// TIA Portal V20 export
FUNCTION_BLOCK "FB_IntLoadUnloadOP"   // FB73, SCL
{ S7_Optimized_Access := 'TRUE' }
// stored: AutoNumber false, MemoryReserve 100, SetENOAutomatically false
   VAR_INPUT
      iStartSeqCond : Bool;   // Start Sequence Conditions
      iJobReq : Bool;   // Job Request - From Main
      iShuttleIntLoadUnloadPos : Bool;   // Load/Unload Pos. Reached - Param
      iShuttleIntLoadUnloadPosSetPoint : LReal;   // Load/Unload Pos. Setpoint - Param
      iShuttleIntLoadUnloadOP_Pos : Bool;   // Load/Unload Pos. Reached - Param
      iShuttleIntLoadUnloadOP_PosSetPoint : LReal;   // Load/Unload Pos. Setpoint - Param
      iAxisV_LoadUnloadShuttlePos : Bool;
      iAxisV_LoadUnloadShuttlePosSetPoint : LReal;
      iAxisV_SafePos : Bool;
      iAxisV_SafePosSetPoint : LReal;
      iAxisW_SafePos : Bool;
      iAxisW_SafePosSetPoint : LReal;
      iAxisW_ApproachLoadUnloadPos : Bool;
      iAxisW_ApproachLoadUnloadSetPoint : LReal;
      iAxisW_LoadUnloadPos : Bool;
      iAxisW_LoadUnloadPosSetPoint : LReal;
      iShuttleMoving : Bool;   // Shuttle is moving - From FB_LoaderAxis
      iShuttleInPos : Bool;   // Shuttle pos. reached - From FB_LoaderAxis
      iAxisV_Moving : Bool;   // Shuttle is moving
      iAxisV_InPos : Bool;
      iAxisW_Moving { ExternalAccessible := 'False'; ExternalVisible := 'False'; ExternalWritable := 'False'} : Bool;   // Shuttle is moving
      iAxisW_InPos : Bool;
      iDrilledPartToUnload : Bool;   // Drilled Part To Unload - From FB_Position
      iUnDrilledPartToLoad : Bool;   // Unrilled Part To Load - From FB_Position
      iLoadGripperClosed : Bool;
      iUnloadGripperOpen : Bool;
      iPLC_DateAndTime : DTL;
      iStepPause : Bool;
   END_VAR
   VAR_OUTPUT
      oShuttleStartReq { ExternalAccessible := 'False'; ExternalVisible := 'False'; ExternalWritable := 'False'} : Bool;   // Shuttle Start Order - To FB_LoaderAxis
      oShuttlePosSetPoint { ExternalAccessible := 'False'; ExternalVisible := 'False'; ExternalWritable := 'False'} : Real;   // Shuttle Position Setpoint - To FB_LoaderAxis
      oAxisV_StartReq : Bool;
      oAxisV_PosSetPoint : Real;
      oAxisW_StartReq : Bool;
      oAxisW_PosSetPoint : Real;
      oLoadGripperCloseReq : Bool;
      oUnloadGripperOpenReq : Bool;
   END_VAR
   VAR
      sCurrent_Step_NB : Int;   // Active Step Number
      sCheck_Step_Condition : Bool;
      sOneStepForward : Bool;
      sRTOneStepForward : R_TRIG;
      sOneStepMode { S7_SetPoint := 'True'} : Bool;
      sStepForward : Bool;
      sInterface : "UDT_SequenceInterface";
      sShuttleStartReq { ExternalAccessible := 'False'; ExternalVisible := 'False'; ExternalWritable := 'False'} : Bool;
      sShuttlePosSetPoint { ExternalAccessible := 'False'; ExternalVisible := 'False'; ExternalWritable := 'False'} : Real;
      sAxisV_StartReq : Bool;
      sAxisV_PosSetPoint : Real;
      sAxisW_StartReq : Bool;
      sAxisW_PosSetPoint : Real;
      sLoadGripperCloseReq : Bool;   // Drilled Part To Unload - From FB_Position
      sUnloadGripperOpenReq : Bool;   // Unrilled Part To Load - From FB_Position
      sTimerAfterGripperClose : TON_TIME;
      sTimerAfterGripperOpen : TON_TIME;
      sTimerAfterApproach { S7_SetPoint := 'True'} : TON_TIME;
      sHistory : Struct
         Activation : Bool;
         Steps : Array[0..99] of Int;
         Date_Time : Array[0..99] of DTL;
      END_STRUCT;
      StepText : "FB_GetTextErrorCode";
   END_VAR
   VAR_TEMP
      tIndex : Int;   // Index
   END_VAR
   VAR CONSTANT
      S00_INIT : Int := 0;
      S10_CHECK_INT_LOAD_UNLOAD_OPTION : Int := 10;
      S20_SHUTTLE_TO_INT_LOAD_UNLOAD_POS_START_REQ : Int := 20;
      S30_SHUTTLE_TO_INT_LOAD_UNLOAD_POS_REACHED : Int := 30;
      S40_AXIS_W_TO_SAFE_POS_START_REQ : Int := 40;
      S50_AXIS_W_TO_SAFE_POS_REACHED : Int := 50;
      S60_AXIS_V_TO_INT_LOAD_UNLOAD_POS_START_REQ : Int := 60;
      S70_AXIS_V_TO_INT_LOAD_UNLOAD_POS_REACHED : Int := 70;
      S80_AXIS_W_TO_INT_LOAD_UNLOAD_APPROACH_POS_START_REQ : Int := 80;
      S90_AXIS_W_TO_INT_LOAD_UNLOAD_APPROACH_POS_REACHED : Int := 90;
      S100_AXIS_W_TO_INT_LOAD_UNLOAD_POS_START_REQ : Int := 100;
      S110_AXIS_W_TO_INT_LOAD_UNLOAD_POS_REACHED : Int := 110;
      S120_CLOSE_LOAD_GRIPPER : Int := 120;
      S130_AXIS_W_TO_SAFE_POS_START_REQ : Int := 130;
      S140_AXIS_W_TO_SAFE_POS_REACHED : Int := 140;
      S150_SHUTTLE_TO_INT_LOAD_UNLOAD_OP_POS_START_REQ : Int := 150;
      S160_SHUTTLE_TO_INT_LOAD_UNLOAD_OP_POS_REACHED : Int := 160;
      S170_AXIS_W_TO_INT_LOAD_UNLOAD_APPROACH_POS_START_REQ : Int := 170;
      S180_AXIS_W_TO_INT_LOAD_UNLOAD_APPROACH_POS_REACHED : Int := 180;
      S190_AXIS_W_TO_INT_LOAD_UNLOAD_POS_START_REQ : Int := 190;
      S200_AXIS_W_TO_INT_LOAD_UNLOAD_POS_REACHED : Int := 200;
      S210_OPEN_UNLOAD_GRIPPER : Int := 210;
      S220_AXIS_W_TO_SAFE_POS_START_REQ : Int := 220;
      S230_AXIS_W_TO_SAFE_POS_REACHED : Int := 230;
      S240_AXIS_V_TO_SAFE_POS_START_REQ : Int := 240;
      S250_AXIS_V_TO_SAFE_POS_REACHED : Int := 250;
      S260_NO_PART_TO_LOAD_UNLOAD : Int := 260;
      S295_JOB_DONE : Int := 295;
   END_VAR
   // StepText.sCode_error[0].ErrorCode := 0;
   // StepText.sCode_error[1].ErrorCode := 10;
   // StepText.sCode_error[2].ErrorCode := 20;
   // StepText.sCode_error[3].ErrorCode := 30;
   // StepText.sCode_error[4].ErrorCode := 40;
   // StepText.sCode_error[5].ErrorCode := 50;
   // StepText.sCode_error[6].ErrorCode := 60;
   // StepText.sCode_error[7].ErrorCode := 70;
   // StepText.sCode_error[8].ErrorCode := 80;
   // StepText.sCode_error[9].ErrorCode := 90;
   // StepText.sCode_error[10].ErrorCode := 95;
BEGIN
   REGION Description header 
       //==================================================================================
       // POSALUX Swiss SA / (C) Copyright 2026
       //----------------------------------------------------------------------------------
       // Title: FB_ExtLoadUnload_OP
       // Comment/Function: 
       // Author: Fabien WALDT
       // Engineering: TIA Portal v20
       //----------------------------------------------------------------------------------
       // Change log table:
       // Version  | Date     | Expert in charge | Changes applied
       // ---------|----------|------------------|-----------------------------------------
       // 00.00.01 | 20260128 | WFA              | First released version
       // =================================================================================
   END_REGION

   REGION Define condition to start
       IF #iStartSeqCond THEN
           #sInterface.SequenceReleased := TRUE;
       ELSE
           // Standard sequencer controls
           #sInterface.SequenceReleased := FALSE;
           #sCurrent_Step_NB := #S00_INIT;
           #sInterface.SequenceRun := FALSE;
           #sInterface.JobDone := FALSE;
           #sCheck_Step_Condition := FALSE;

           // Dedicated sequencer controls
           #sShuttleStartReq := FALSE;
           #sShuttlePosSetPoint := 0.0;
           #sAxisV_StartReq := FALSE;
           #sAxisV_PosSetPoint := 0.0;
           #sAxisW_StartReq := FALSE;
           #sAxisW_PosSetPoint := 0.0;
           #sLoadGripperCloseReq := FALSE;
           #sUnloadGripperOpenReq := FALSE;

           // Add specifics controls 
       END_IF;

       // Reset interface error
       IF #sInterface.Reset THEN
           #sInterface.Error := FALSE;
       END_IF;

       // Reset start when axis in position
       IF #iShuttleInPos THEN
           #sShuttleStartReq := FALSE;
       END_IF;
       IF #iAxisV_InPos THEN
           #sAxisV_StartReq := FALSE;
       END_IF;
       IF #iAxisW_InPos THEN
           #sAxisW_StartReq := FALSE;
       END_IF;

       // One step forward
       #sRTOneStepForward.CLK := #sOneStepForward;
       #sRTOneStepForward();
       #sStepForward := (NOT #sOneStepMode OR (#sOneStepMode AND #sRTOneStepForward.Q)) AND NOT #iStepPause;
       #sOneStepForward := FALSE;

       // Action only true in dedicated steps
       #sLoadGripperCloseReq := FALSE;
       #sUnloadGripperOpenReq := FALSE;

       // Timer Gripper OK
       #"sTimerAfterGripperClose"(IN := #sCurrent_Step_NB = 120
                                  AND ((#iUnDrilledPartToLoad AND #iLoadGripperClosed) OR NOT #iUnDrilledPartToLoad),
                                  PT := T#500ms);
       #"sTimerAfterGripperOpen"(IN := #sCurrent_Step_NB = 210
                                 AND ((#iDrilledPartToUnload AND #iUnloadGripperOpen) OR NOT #iDrilledPartToUnload),
                                 PT := T#500ms);

       // Timer between approach and Load/Unload position
       #sTimerAfterApproach(IN := (#sCurrent_Step_NB = 90 OR #sCurrent_Step_NB = 180) AND #iAxisW_ApproachLoadUnloadPos,
                            PT := T#100ms);
   END_REGION

   REGION Sequence Function
       CASE #sCurrent_Step_NB OF
           #S00_INIT:
               REGION S00 INIT
                   #sCheck_Step_Condition := TRUE;
               END_REGION
           #S10_CHECK_INT_LOAD_UNLOAD_OPTION:
               REGION S10_CHECK_INT_LOAD_UNLOAD_OPTION
                   #sCheck_Step_Condition := TRUE;
               END_REGION
           #S20_SHUTTLE_TO_INT_LOAD_UNLOAD_POS_START_REQ:
               REGION S20_SHUTTLE_TO_INT_LOAD_UNLOAD_POS_START_REQ
                   #sShuttleStartReq := NOT #iShuttleIntLoadUnloadPos;
                   #sShuttlePosSetPoint := LREAL_TO_REAL(#iShuttleIntLoadUnloadPosSetPoint);
                   #sCheck_Step_Condition := TRUE;
               END_REGION
           #S30_SHUTTLE_TO_INT_LOAD_UNLOAD_POS_REACHED:
               REGION S30_SHUTTLE_TO_INT_LOAD_UNLOAD_POS_REACHED
                   #sCheck_Step_Condition := TRUE;
               END_REGION
           #S40_AXIS_W_TO_SAFE_POS_START_REQ:
               REGION S40_AXIS_W_TO_SAFE_POS_START_REQ
                   #sAxisW_StartReq := NOT #iAxisW_SafePos;
                   #sAxisW_PosSetPoint := LREAL_TO_REAL(#iAxisW_SafePosSetPoint);
                   #sCheck_Step_Condition := TRUE;
               END_REGION
           #S50_AXIS_W_TO_SAFE_POS_REACHED:
               REGION S50_AXIS_W_TO_SAFE_POS_REACHED
                   #sCheck_Step_Condition := TRUE;
               END_REGION
           #S60_AXIS_V_TO_INT_LOAD_UNLOAD_POS_START_REQ:
               REGION S60_AXIS_V_TO_INT_LOAD_UNLOAD_POS_START_REQ
                   #sAxisV_StartReq := NOT #iAxisV_LoadUnloadShuttlePos;
                   #sAxisV_PosSetPoint := LREAL_TO_REAL(#iAxisV_LoadUnloadShuttlePosSetPoint);
                       #sCheck_Step_Condition := TRUE;
                   END_REGION
           #S70_AXIS_V_TO_INT_LOAD_UNLOAD_POS_REACHED:
               REGION S70_AXIS_V_TO_INT_LOAD_UNLOAD_POS_REACHED
                   #sCheck_Step_Condition := TRUE;
               END_REGION
           #S80_AXIS_W_TO_INT_LOAD_UNLOAD_APPROACH_POS_START_REQ:
               REGION S80_AXIS_W_TO_INT_LOAD_UNLOAD_APPROACH_POS_START_REQ
                   #sAxisW_StartReq := NOT #iAxisW_ApproachLoadUnloadPos;
                   #sAxisW_PosSetPoint := LREAL_TO_REAL(#iAxisW_ApproachLoadUnloadSetPoint);
                   #sCheck_Step_Condition := TRUE;
               END_REGION
           #S90_AXIS_W_TO_INT_LOAD_UNLOAD_APPROACH_POS_REACHED:
               REGION S90_AXIS_W_TO_INT_LOAD_UNLOAD_APPROACH_POS_REACHED
                   IF #sTimerAfterApproach.Q THEN
                       #sCheck_Step_Condition := TRUE;
                   END_IF;
               END_REGION
           #S100_AXIS_W_TO_INT_LOAD_UNLOAD_POS_START_REQ:
               REGION S100_AXIS_W_TO_INT_LOAD_UNLOAD_POS_START_REQ
                   #sAxisW_StartReq := NOT #iAxisW_LoadUnloadPos;
                   #sAxisW_PosSetPoint := LREAL_TO_REAL(#iAxisW_LoadUnloadPosSetPoint);
                   #sCheck_Step_Condition := TRUE;
               END_REGION
           #S110_AXIS_W_TO_INT_LOAD_UNLOAD_POS_REACHED:
               REGION S110_AXIS_W_TO_INT_LOAD_UNLOAD_POS_REACHED
                   #sCheck_Step_Condition := TRUE;
               END_REGION
           #S120_CLOSE_LOAD_GRIPPER:
               REGION S120_CLOSE_LOAD_GRIPPER
                   #sLoadGripperCloseReq := #iUnDrilledPartToLoad;
                   IF #"sTimerAfterGripperClose".Q THEN
                       #sCheck_Step_Condition := TRUE;
                   END_IF;
               END_REGION
           #S130_AXIS_W_TO_SAFE_POS_START_REQ:
               REGION S130_AXIS_W_TO_SAFE_POS_START_REQ
                   #sAxisW_StartReq := NOT #iAxisW_SafePos;
                   #sAxisW_PosSetPoint := LREAL_TO_REAL(#iAxisW_SafePosSetPoint);
                   #sCheck_Step_Condition := TRUE;
               END_REGION
           #S140_AXIS_W_TO_SAFE_POS_REACHED:
               REGION S140_AXIS_W_TO_SAFE_POS_REACHED
                   #sCheck_Step_Condition := TRUE;
               END_REGION
           #S150_SHUTTLE_TO_INT_LOAD_UNLOAD_OP_POS_START_REQ:
               REGION S150_SHUTTLE_TO_INT_LOAD_UNLOAD_OP_POS_START_REQ
                   #sShuttleStartReq := NOT #iShuttleIntLoadUnloadOP_Pos;
                   #sShuttlePosSetPoint := LREAL_TO_REAL(#iShuttleIntLoadUnloadOP_PosSetPoint);
                   #sCheck_Step_Condition := TRUE;
               END_REGION
           #S160_SHUTTLE_TO_INT_LOAD_UNLOAD_OP_POS_REACHED:
               REGION S160_SHUTTLE_TO_INT_LOAD_UNLOAD_OP_POS_REACHED
                   #sCheck_Step_Condition := TRUE;
               END_REGION
           #S170_AXIS_W_TO_INT_LOAD_UNLOAD_APPROACH_POS_START_REQ:
               REGION S170_AXIS_W_TO_INT_LOAD_UNLOAD_APPROACH_POS_START_REQ
                   #sAxisW_StartReq := NOT #iAxisW_ApproachLoadUnloadPos;
                   #sAxisW_PosSetPoint := LREAL_TO_REAL(#iAxisW_ApproachLoadUnloadSetPoint);
                   #sCheck_Step_Condition := TRUE;
               END_REGION
           #S180_AXIS_W_TO_INT_LOAD_UNLOAD_APPROACH_POS_REACHED:
               REGION S180_AXIS_W_TO_INT_LOAD_UNLOAD_APPROACH_POS_REACHED
                   IF #sTimerAfterApproach.Q THEN
                       #sCheck_Step_Condition := TRUE;
                   END_IF;
               END_REGION
           #S190_AXIS_W_TO_INT_LOAD_UNLOAD_POS_START_REQ:
               REGION S190_AXIS_W_TO_INT_LOAD_UNLOAD_POS_START_REQ
                   #sAxisW_StartReq := NOT #iAxisW_LoadUnloadPos;
                   #sAxisW_PosSetPoint := LREAL_TO_REAL(#iAxisW_LoadUnloadPosSetPoint);
                   #sCheck_Step_Condition := TRUE;
               END_REGION
           #S200_AXIS_W_TO_INT_LOAD_UNLOAD_POS_REACHED:
               REGION S200_AXIS_W_TO_INT_LOAD_UNLOAD_POS_REACHED
                   #sCheck_Step_Condition := TRUE;
               END_REGION
           #S210_OPEN_UNLOAD_GRIPPER:
               REGION S210_OPEN_UNLOAD_GRIPPER
                   #sUnloadGripperOpenReq := #iDrilledPartToUnload;
                   IF #"sTimerAfterGripperOpen".Q THEN
                       #sCheck_Step_Condition := TRUE;
                   END_IF;
               END_REGION
           #S220_AXIS_W_TO_SAFE_POS_START_REQ:
               REGION S220_AXIS_W_TO_SAFE_POS_START_REQ
                   #sAxisW_StartReq := NOT #iAxisW_SafePos;
                   #sAxisW_PosSetPoint := LREAL_TO_REAL(#iAxisW_SafePosSetPoint);
                   #sCheck_Step_Condition := TRUE;
               END_REGION
           #S230_AXIS_W_TO_SAFE_POS_REACHED:
               REGION S230_AXIS_W_TO_SAFE_POS_REACHED
                   #sCheck_Step_Condition := TRUE;
               END_REGION
           #S240_AXIS_V_TO_SAFE_POS_START_REQ:
               REGION S240_AXIS_V_TO_SAFE_POS_START_REQ
                   #sAxisV_StartReq := NOT #iAxisV_SafePos;
                   #sAxisV_PosSetPoint := LREAL_TO_REAL(#iAxisV_SafePosSetPoint);
                   #sCheck_Step_Condition := TRUE;
               END_REGION
           #S250_AXIS_V_TO_SAFE_POS_REACHED:
               REGION S250_AXIS_V_TO_SAFE_POS_REACHED
                   #sCheck_Step_Condition := TRUE;
               END_REGION
           #S260_NO_PART_TO_LOAD_UNLOAD:
               REGION S260_NO_PART_TO_LOAD_UNLOAD
                   #sCheck_Step_Condition := TRUE;
               END_REGION
           #S295_JOB_DONE:
               REGION S295_JOB_DONE
                   #sInterface.JobDone := TRUE;
                   #sCheck_Step_Condition := TRUE;
               END_REGION
           ELSE:
               #sInterface.Error := TRUE;
       END_CASE;
   END_REGION

   REGION Sequence Next Step Condition
       IF #sCheck_Step_Condition THEN
           CASE #sCurrent_Step_NB OF
               #S00_INIT:
                   REGION S00 INIT
                       IF #sInterface.SequenceReleased AND #iJobReq THEN
                           #sCurrent_Step_NB := #S10_CHECK_INT_LOAD_UNLOAD_OPTION;
                           #sInterface.SequenceRun := TRUE;
                           #sCheck_Step_Condition := FALSE;
                       ELSE
                           #sInterface.SequenceRun := FALSE;
                       END_IF;
                   END_REGION
               #S10_CHECK_INT_LOAD_UNLOAD_OPTION:
                   REGION S10_CHECK_INT_LOAD_UNLOAD_OPTION
                       IF #sInterface.SequenceReleased AND #sStepForward AND "DB_LoaderOptions".IntLoadUnload.CommonPos AND (#iDrilledPartToUnload OR #iUnDrilledPartToLoad) THEN
                           #sCurrent_Step_NB := #S20_SHUTTLE_TO_INT_LOAD_UNLOAD_POS_START_REQ;
                           #sCheck_Step_Condition := FALSE;
                       ELSIF #sInterface.SequenceReleased AND #sStepForward AND "DB_LoaderOptions".IntLoadUnload.CommonPos AND NOT #iJobReq OR (NOT #iDrilledPartToUnload AND NOT #iUnDrilledPartToLoad) THEN
                           #sCurrent_Step_NB := #S260_NO_PART_TO_LOAD_UNLOAD;
                           #sCheck_Step_Condition := FALSE;
                       END_IF;
                   END_REGION
               #S20_SHUTTLE_TO_INT_LOAD_UNLOAD_POS_START_REQ:
                   REGION S20_SHUTTLE_TO_INT_LOAD_UNLOAD_POS_START_REQ
                       IF #sInterface.SequenceReleased AND (#iShuttleMoving OR #iShuttleIntLoadUnloadPos) THEN
                           #sCurrent_Step_NB := #S30_SHUTTLE_TO_INT_LOAD_UNLOAD_POS_REACHED;
                           #sCheck_Step_Condition := FALSE;
                       END_IF;
                   END_REGION
               #S30_SHUTTLE_TO_INT_LOAD_UNLOAD_POS_REACHED:
                   REGION S30_SHUTTLE_TO_INT_LOAD_UNLOAD_POS_REACHED
                       IF #sInterface.SequenceReleased AND #sStepForward AND NOT #sShuttleStartReq AND #iShuttleIntLoadUnloadPos THEN
                           #sCurrent_Step_NB := #S60_AXIS_V_TO_INT_LOAD_UNLOAD_POS_START_REQ;
                           #sCheck_Step_Condition := FALSE;
                       END_IF;
                   END_REGION
               #S40_AXIS_W_TO_SAFE_POS_START_REQ:
                   REGION S40_AXIS_W_TO_SAFE_POS_START_REQ
                       IF #sInterface.SequenceReleased AND #sStepForward AND (#iAxisW_Moving OR #iAxisW_SafePos) THEN
                           #sCurrent_Step_NB := #S50_AXIS_W_TO_SAFE_POS_REACHED;
                           #sCheck_Step_Condition := FALSE;
                       END_IF;
                   END_REGION
               #S50_AXIS_W_TO_SAFE_POS_REACHED:
                   REGION S50_AXIS_W_TO_SAFE_POS_REACHED
                       IF #sInterface.SequenceReleased AND #sStepForward AND NOT #sAxisW_StartReq AND #iAxisW_SafePos THEN
                           #sCurrent_Step_NB := #S60_AXIS_V_TO_INT_LOAD_UNLOAD_POS_START_REQ;
                           #sCheck_Step_Condition := FALSE;
                       END_IF;
                   END_REGION
               #S60_AXIS_V_TO_INT_LOAD_UNLOAD_POS_START_REQ:
                   REGION S60_AXIS_V_TO_INT_LOAD_UNLOAD_POS_START_REQ
                       IF #sInterface.SequenceReleased AND (#iAxisV_Moving OR #iAxisV_LoadUnloadShuttlePos) THEN
                           #sCurrent_Step_NB := #S70_AXIS_V_TO_INT_LOAD_UNLOAD_POS_REACHED;
                           #sCheck_Step_Condition := FALSE;
                       END_IF;
                   END_REGION
               #S70_AXIS_V_TO_INT_LOAD_UNLOAD_POS_REACHED:
                   REGION S70_AXIS_V_TO_INT_LOAD_UNLOAD_POS_REACHED
                       IF #sInterface.SequenceReleased AND #sStepForward AND NOT #sAxisV_StartReq AND #iAxisV_LoadUnloadShuttlePos THEN
                           #sCurrent_Step_NB := #S80_AXIS_W_TO_INT_LOAD_UNLOAD_APPROACH_POS_START_REQ;
                           #sCheck_Step_Condition := FALSE;
                       END_IF;
                   END_REGION
               #S80_AXIS_W_TO_INT_LOAD_UNLOAD_APPROACH_POS_START_REQ:
                   REGION S80_AXIS_W_TO_INT_LOAD_UNLOAD_APPROACH_POS_START_REQ
                       IF #sInterface.SequenceReleased AND (#iAxisW_Moving OR #iAxisW_ApproachLoadUnloadPos) THEN
                           #sCurrent_Step_NB := #S90_AXIS_W_TO_INT_LOAD_UNLOAD_APPROACH_POS_REACHED;
                           #sCheck_Step_Condition := FALSE;
                       END_IF;
                   END_REGION
               #S90_AXIS_W_TO_INT_LOAD_UNLOAD_APPROACH_POS_REACHED:
                   REGION S90_AXIS_W_TO_INT_LOAD_UNLOAD_APPROACH_POS_REACHED
                       IF #sInterface.SequenceReleased AND #sStepForward AND NOT #sAxisW_StartReq AND #iAxisW_ApproachLoadUnloadPos THEN
                           #sCurrent_Step_NB := #S100_AXIS_W_TO_INT_LOAD_UNLOAD_POS_START_REQ;
                           #sCheck_Step_Condition := FALSE;
                       END_IF;
                   END_REGION
               #S100_AXIS_W_TO_INT_LOAD_UNLOAD_POS_START_REQ:
                   REGION S100_AXIS_W_TO_INT_LOAD_UNLOAD_POS_START_REQ
                       IF #sInterface.SequenceReleased AND (#iAxisW_Moving OR #iAxisW_LoadUnloadPos) THEN
                           #sCurrent_Step_NB := #S110_AXIS_W_TO_INT_LOAD_UNLOAD_POS_REACHED;
                           #sCheck_Step_Condition := FALSE;
                       END_IF;
                   END_REGION
               #S110_AXIS_W_TO_INT_LOAD_UNLOAD_POS_REACHED:
                   REGION S110_AXIS_W_TO_INT_LOAD_UNLOAD_POS_REACHED
                       IF #sInterface.SequenceReleased AND #sStepForward AND NOT #sAxisW_StartReq AND #iAxisW_LoadUnloadPos THEN
                           #sCurrent_Step_NB := #S120_CLOSE_LOAD_GRIPPER;
                           #sCheck_Step_Condition := FALSE;
                       END_IF;
                   END_REGION
               #S120_CLOSE_LOAD_GRIPPER:
                   REGION S120_CLOSE_LOAD_GRIPPER
                       IF #sInterface.SequenceReleased AND #sStepForward
                           AND ((#iUnDrilledPartToLoad AND #iLoadGripperClosed) OR NOT #iUnDrilledPartToLoad) THEN
                           #sCurrent_Step_NB := #S130_AXIS_W_TO_SAFE_POS_START_REQ;
                           #sCheck_Step_Condition := FALSE;
                       END_IF;
                   END_REGION
               #S130_AXIS_W_TO_SAFE_POS_START_REQ:
                   REGION S130_AXIS_W_TO_SAFE_POS_START_REQ
                       IF #sInterface.SequenceReleased AND (#iAxisW_Moving OR #iAxisW_SafePos) THEN
                           #sCurrent_Step_NB := #S140_AXIS_W_TO_SAFE_POS_REACHED;
                           #sCheck_Step_Condition := FALSE;
                       END_IF;
                   END_REGION
               #S140_AXIS_W_TO_SAFE_POS_REACHED:
                   REGION S140_AXIS_W_TO_SAFE_POS_REACHED
                       IF #sInterface.SequenceReleased AND #sStepForward AND NOT #sAxisW_StartReq AND #iAxisW_SafePos THEN
                           #sCurrent_Step_NB := #S150_SHUTTLE_TO_INT_LOAD_UNLOAD_OP_POS_START_REQ;
                           #sCheck_Step_Condition := FALSE;
                       END_IF;
                   END_REGION
               #S150_SHUTTLE_TO_INT_LOAD_UNLOAD_OP_POS_START_REQ:
                   REGION S150_SHUTTLE_TO_INT_LOAD_UNLOAD_OP_POS_START_REQ
                       IF #sInterface.SequenceReleased AND (#iShuttleMoving OR #iShuttleIntLoadUnloadOP_Pos) THEN
                           #sCurrent_Step_NB := #S160_SHUTTLE_TO_INT_LOAD_UNLOAD_OP_POS_REACHED;
                           #sCheck_Step_Condition := FALSE;
                       END_IF;
                   END_REGION
               #S160_SHUTTLE_TO_INT_LOAD_UNLOAD_OP_POS_REACHED:
                   REGION S160_SHUTTLE_TO_INT_LOAD_UNLOAD_OP_POS_REACHED
                       IF #sInterface.SequenceReleased AND #sStepForward AND NOT #sShuttleStartReq AND #iShuttleIntLoadUnloadOP_Pos THEN
                           #sCurrent_Step_NB := #S170_AXIS_W_TO_INT_LOAD_UNLOAD_APPROACH_POS_START_REQ;
                           #sCheck_Step_Condition := FALSE;
                       END_IF;
                   END_REGION
               #S170_AXIS_W_TO_INT_LOAD_UNLOAD_APPROACH_POS_START_REQ:
                   REGION S170_AXIS_W_TO_INT_LOAD_UNLOAD_APPROACH_POS_START_REQ
                       IF #sInterface.SequenceReleased AND (#iAxisW_Moving OR #iAxisW_ApproachLoadUnloadPos) THEN
                           #sCurrent_Step_NB := #S180_AXIS_W_TO_INT_LOAD_UNLOAD_APPROACH_POS_REACHED;
                           #sCheck_Step_Condition := FALSE;
                       END_IF;
                   END_REGION
               #S180_AXIS_W_TO_INT_LOAD_UNLOAD_APPROACH_POS_REACHED:
                   REGION S180_AXIS_W_TO_INT_LOAD_UNLOAD_APPROACH_POS_REACHED
                       IF #sInterface.SequenceReleased AND #sStepForward AND NOT #sAxisW_StartReq AND #iAxisW_ApproachLoadUnloadPos THEN
                           #sCurrent_Step_NB := #S190_AXIS_W_TO_INT_LOAD_UNLOAD_POS_START_REQ;
                           #sCheck_Step_Condition := FALSE;
                       END_IF;
                   END_REGION
               #S190_AXIS_W_TO_INT_LOAD_UNLOAD_POS_START_REQ:
                   REGION S190_AXIS_W_TO_INT_LOAD_UNLOAD_POS_START_REQ
                       IF #sInterface.SequenceReleased AND (#iAxisW_Moving OR #iAxisW_LoadUnloadPos) THEN
                           #sCurrent_Step_NB := #S200_AXIS_W_TO_INT_LOAD_UNLOAD_POS_REACHED;
                           #sCheck_Step_Condition := FALSE;
                       END_IF;
                   END_REGION
               #S200_AXIS_W_TO_INT_LOAD_UNLOAD_POS_REACHED:
                   REGION S200_AXIS_W_TO_INT_LOAD_UNLOAD_POS_REACHED
                       IF #sInterface.SequenceReleased AND #sStepForward AND NOT #sAxisW_StartReq AND #iAxisW_LoadUnloadPos THEN
                           #sCurrent_Step_NB := #S210_OPEN_UNLOAD_GRIPPER;
                           #sCheck_Step_Condition := FALSE;
                       END_IF;
                   END_REGION
               #S210_OPEN_UNLOAD_GRIPPER:
                   REGION S210_OPEN_UNLOAD_GRIPPER
                       IF #sInterface.SequenceReleased AND #sStepForward
                           AND (#iDrilledPartToUnload AND #iUnloadGripperOpen OR NOT #iDrilledPartToUnload) THEN
                           #sCurrent_Step_NB := #S220_AXIS_W_TO_SAFE_POS_START_REQ;
                           #sCheck_Step_Condition := FALSE;
                       END_IF;
                   END_REGION
               #S220_AXIS_W_TO_SAFE_POS_START_REQ:
                   REGION S220_AXIS_W_TO_SAFE_POS_START_REQ
                       IF #sInterface.SequenceReleased AND (#iAxisW_Moving OR #iAxisW_SafePos) THEN
                           #sCurrent_Step_NB := #S230_AXIS_W_TO_SAFE_POS_REACHED;
                           #sCheck_Step_Condition := FALSE;
                       END_IF;
                   END_REGION
               #S230_AXIS_W_TO_SAFE_POS_REACHED:
                   REGION S230_AXIS_W_TO_SAFE_POS_REACHED
                       IF #sInterface.SequenceReleased AND #sStepForward AND NOT #sAxisW_StartReq AND #iAxisW_SafePos THEN
                           #sCurrent_Step_NB := #S295_JOB_DONE;
                           #sCheck_Step_Condition := FALSE;
                       END_IF;
                   END_REGION
               #S240_AXIS_V_TO_SAFE_POS_START_REQ:
                   REGION S240_AXIS_V_TO_SAFE_POS_START_REQ
                       IF #sInterface.SequenceReleased AND (#iAxisV_Moving OR #iAxisV_SafePos) THEN
                           #sCurrent_Step_NB := #S250_AXIS_V_TO_SAFE_POS_REACHED;
                           #sCheck_Step_Condition := FALSE;
                       END_IF;
                   END_REGION
               #S250_AXIS_V_TO_SAFE_POS_REACHED:
                   REGION S160_AXIS_V_TO_SAFE_POS_REACHED
                       IF #sInterface.SequenceReleased AND #sStepForward AND NOT #sAxisV_StartReq AND #iAxisV_SafePos THEN
                           #sCurrent_Step_NB := #S295_JOB_DONE;
                           #sCheck_Step_Condition := FALSE;
                       END_IF;
                   END_REGION
               #S260_NO_PART_TO_LOAD_UNLOAD:
                   REGION S260_NO_PART_TO_LOAD_UNLOAD
                       IF #sInterface.SequenceReleased AND #sStepForward AND "AlwaysTRUE" THEN
                           #sCurrent_Step_NB := #S220_AXIS_W_TO_SAFE_POS_START_REQ;
                           #sCheck_Step_Condition := FALSE;
                       END_IF;
                   END_REGION
               #S295_JOB_DONE:
                   REGION S95_JOB_DONE
                       IF NOT #iJobReq THEN
                           #sCurrent_Step_NB := #S00_INIT;
                           #sCheck_Step_Condition := FALSE;
                           #sInterface.JobDone := FALSE;
                       END_IF;
                   END_REGION
               ELSE
                   #sInterface.Error := TRUE;
           END_CASE;
       END_IF;
   END_REGION

   REGION Outputs Update
       #oShuttleStartReq := #sShuttleStartReq;
       #oShuttlePosSetPoint := #sShuttlePosSetPoint;
       #oAxisV_StartReq := #sAxisV_StartReq;
       #oAxisV_PosSetPoint := #sAxisV_PosSetPoint;
       #oAxisW_StartReq := #sAxisW_StartReq;
       #oAxisW_PosSetPoint := #sAxisW_PosSetPoint;
       #oLoadGripperCloseReq := #sLoadGripperCloseReq;
       #oUnloadGripperOpenReq := #sUnloadGripperOpenReq;

   END_REGION

   REGION Steps - Date and Time History
       IF #sHistory.Activation THEN
           IF #sHistory.Steps[0] <> #sCurrent_Step_NB THEN
               FOR #tIndex := 98 TO 0 BY -1 DO
                   #sHistory.Steps[#tIndex + 1] := #sHistory.Steps[#tIndex];
                   #sHistory.Date_Time[#tIndex + 1] := #sHistory.Date_Time[#tIndex];
               END_FOR;
               #sHistory.Steps[0] := #sCurrent_Step_NB;
               #sHistory.Date_Time[0] := #iPLC_DateAndTime;
           END_IF;
       END_IF;
   END_REGION

   REGION Steps Text
       #StepText(iErrorCode := #sCurrent_Step_NB,
                 oErrorText => #StepText.oErrorText);
   END_REGION
END_FUNCTION_BLOCK
